SUBAPPLICATION Schneidwerk (* Subapplication Type *)
  (* Standard: 61499-2 *)
  (* Version 1.0, 2023-01-29, Franz *)
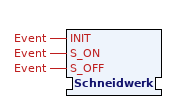
  EVENT_INPUT
    INIT;
    S_ON;
    S_OFF;
  END_EVENT
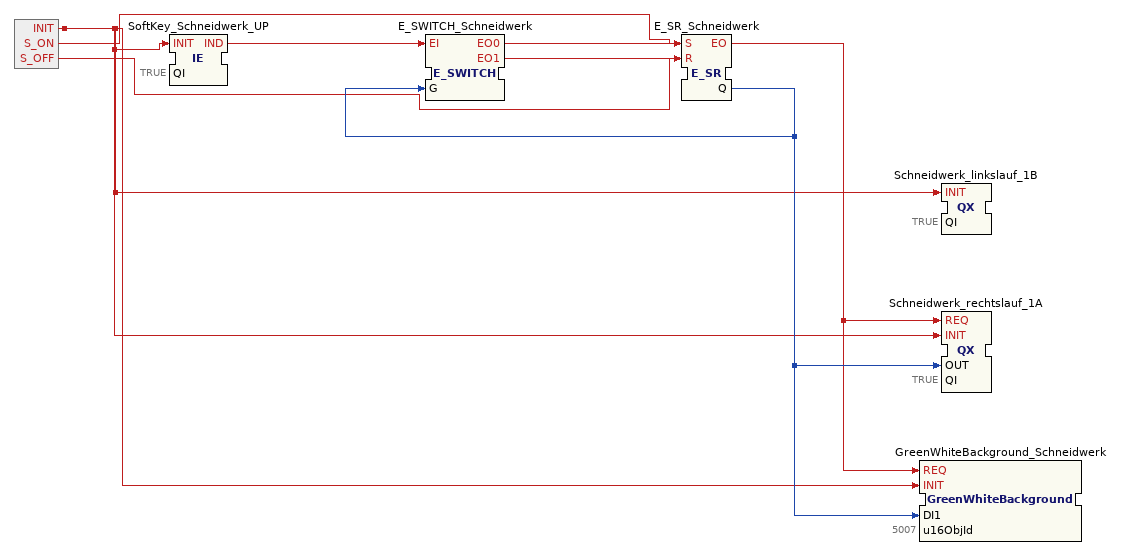
  FBS
    Schneidwerk_rechtslauf_1A : QX(QI := TRUE);
    GreenWhiteBackground_Schneidwerk : GreenWhiteBackground(u16ObjId := 5007);
    E_SWITCH_Schneidwerk : E_SWITCH;
    E_SR_Schneidwerk : E_SR;
    Schneidwerk_linkslauf_1B : QX(QI := TRUE);
    SoftKey_Schneidwerk_UP : IE(QI := TRUE);
  END_FBS
  EVENT_CONNECTIONS
    E_SR_Schneidwerk.EO TO Schneidwerk_rechtslauf_1A.REQ;
    E_SR_Schneidwerk.EO TO GreenWhiteBackground_Schneidwerk.REQ;
    E_SWITCH_Schneidwerk.EO0 TO E_SR_Schneidwerk.S;
    E_SWITCH_Schneidwerk.EO1 TO E_SR_Schneidwerk.R;
    S_ON TO E_SR_Schneidwerk.S;
    S_OFF TO E_SR_Schneidwerk.R;
    INIT TO Schneidwerk_linkslauf_1B.INIT;
    INIT TO GreenWhiteBackground_Schneidwerk.INIT;
    INIT TO Schneidwerk_rechtslauf_1A.INIT;
    INIT TO SoftKey_Schneidwerk_UP.INIT;
    SoftKey_Schneidwerk_UP.IND TO E_SWITCH_Schneidwerk.EI;
  END_CONNECTIONS
  DATA_CONNECTIONS
    E_SR_Schneidwerk.Q TO Schneidwerk_rechtslauf_1A.OUT;
    E_SR_Schneidwerk.Q TO GreenWhiteBackground_Schneidwerk.DI1;
    E_SR_Schneidwerk.Q TO E_SWITCH_Schneidwerk.G;
  END_CONNECTIONS
END_SUBAPPLICATION
